(* IEC 61131-3 sources: MotionTestBenchMaster/Logical/02_HMI/HMI, 4 files *)

(* ---- Counter_Mng.st ---- *)
ACTION HMI_CounterInit:
	HMI_CounterCfgPartial.MachineCounters.HmiData[FillerLaps].Description				:= '@CounterDescription_001';
	HMI_CounterCfgPartial.MachineCounters.HmiData[ClosingUnit1Laps].Description			:= '@CounterDescription_002';
	HMI_CounterCfgPartial.MachineCounters.HmiData[ClosingUnit2Laps].Description			:= '@CounterDescription_003';
	HMI_CounterCfgPartial.MachineCounters.HmiData[RinserLaps].Description				:= '@CounterDescription_004';
	HMI_CounterCfgPartial.MachineCounters.HmiData[FlaworDoserLaps].Description			:= '@CounterDescription_005';
	HMI_CounterCfgPartial.MachineCounters.HmiData[PulpDoserLaps].Description			:= '@CounterDescription_006';
	HMI_CounterCfgPartial.MachineCounters.HmiData[PowerOn].Description					:= '@CounterDescription_007';

	HMI_CounterCfgPartial.ContainersCounters.HmiData[FillingFault].Description			:= '@CounterDescription_008';
	HMI_CounterCfgPartial.ContainersCounters.HmiData[FillingBurst].Description			:= '@CounterDescription_009';
	HMI_CounterCfgPartial.ContainersCounters.HmiData[ClosingUnit1Fault].Description		:= '@CounterDescription_010';
	HMI_CounterCfgPartial.ContainersCounters.HmiData[ClosingUnit2Fault].Description		:= '@CounterDescription_011';
	HMI_CounterCfgPartial.ContainersCounters.HmiData[RinsingFault].Description			:= '@CounterDescription_012';
	HMI_CounterCfgPartial.ContainersCounters.HmiData[PulpDoserFault].Description		:= '@CounterDescription_013';
	HMI_CounterCfgPartial.ContainersCounters.HmiData[FlaworDoserFault].Description		:= '@CounterDescription_014';
	HMI_CounterCfgPartial.ContainersCounters.HmiData[BurstEjected].Description			:= '@CounterDescription_015';
	HMI_CounterCfgPartial.ContainersCounters.HmiData[ManualEjected].Description			:= '@CounterDescription_016';
	HMI_CounterCfgPartial.ContainersCounters.HmiData[LowFillingEjected].Description		:= '@CounterDescription_017';
	HMI_CounterCfgPartial.ContainersCounters.HmiData[NotFilledEjected].Description		:= '@CounterDescription_018';
	HMI_CounterCfgPartial.ContainersCounters.HmiData[ContainersEntered].Description		:= '@CounterDescription_019';
	HMI_CounterCfgPartial.ContainersCounters.HmiData[ContainersProduced].Description	:= '@CounterDescription_020';
	HMI_CounterCfgPartial.ContainersCounters.HmiData[EjectionBySIS].Description			:= '@CounterDescription_045'; //V4.A.A.1.6.8
	HMI_CounterCfgPartial.ContainersCounters.HmiData[SIS_EjectionToBlower].Description			 := '@CounterDescription_046'; //V4.A.A.1.6.8
	HMI_CounterCfgPartial.ContainersCounters.HmiData[SIS_ContainersProducedToBlower].Description := '@CounterDescription_047'; //V4.A.A.1.6.8

	HMI_CounterCfgPartial.ProcessCounters.HmiData[FillerProduction].Description			:= '@CounterDescription_021';
	HMI_CounterCfgPartial.ProcessCounters.HmiData[ClosingUnit1Production].Description	:= '@CounterDescription_022';
	HMI_CounterCfgPartial.ProcessCounters.HmiData[ClosingUnit2Production].Description	:= '@CounterDescription_023';
	HMI_CounterCfgPartial.ProcessCounters.HmiData[RinserProduction].Description			:= '@CounterDescription_024';
	HMI_CounterCfgPartial.ProcessCounters.HmiData[PulpDoserProduction].Description		:= '@CounterDescription_025';
	HMI_CounterCfgPartial.ProcessCounters.HmiData[FlaworDoserProduction].Description	:= '@CounterDescription_026';
	HMI_CounterCfgPartial.ProcessCounters.HmiData[Cop].Description						:= '@CounterDescription_027';
	HMI_CounterCfgPartial.ProcessCounters.HmiData[FillerCip].Description				:= '@CounterDescription_044';
	HMI_CounterCfgPartial.ProcessCounters.HmiData[ClosingUnit1Cip].Description			:= '@CounterDescription_028';
	HMI_CounterCfgPartial.ProcessCounters.HmiData[ClosingUnit2Cip].Description			:= '@CounterDescription_029';
	HMI_CounterCfgPartial.ProcessCounters.HmiData[RinserCip].Description				:= '@CounterDescription_030';
	HMI_CounterCfgPartial.ProcessCounters.HmiData[PulpDoserCip].Description				:= '@CounterDescription_031';
	HMI_CounterCfgPartial.ProcessCounters.HmiData[FlaworDoserCip].Description			:= '@CounterDescription_032';

	HMI_CounterCfgPartial.EcoCounters.HmiData[Power].Description						:= '@CounterDescription_033';
	HMI_CounterCfgPartial.EcoCounters.HmiData[Air].Description							:= '@CounterDescription_034';
	HMI_CounterCfgPartial.EcoCounters.HmiData[GeneralCO2].Description					:= '@CounterDescription_035';
	HMI_CounterCfgPartial.EcoCounters.HmiData[ClosingUnitCO2].Description				:= '@CounterDescription_036';
	HMI_CounterCfgPartial.EcoCounters.HmiData[N2].Description							:= '@CounterDescription_037';
	HMI_CounterCfgPartial.EcoCounters.HmiData[ProcessWater].Description					:= '@CounterDescription_038';
	HMI_CounterCfgPartial.EcoCounters.HmiData[CopWater].Description						:= '@CounterDescription_039';
	HMI_CounterCfgPartial.EcoCounters.HmiData[BottomBottleCoolingWater].Description		:= '@CounterDescription_040';
	HMI_CounterCfgPartial.EcoCounters.HmiData[Product].Description						:= '@CounterDescription_041';
	HMI_CounterCfgPartial.EcoCounters.HmiData[Steam].Description						:= '@CounterDescription_042';
	HMI_CounterCfgPartial.EcoCounters.HmiData[FoodSteam].Description					:= '@CounterDescription_043';
	HMI_CounterCfgPartial.EcoCounters.HmiData[ProductWater].Description					:= '@CounterDescription_049'; //V4.A.A.1.6.14k
	HMI_CounterCfgPartial.EcoCounters.HmiData[Syrup].Description						:= '@CounterDescription_050'; //V4.A.A.1.6.14k

	HMI_CounterCfgPartial.EcoCounters.HmiData[Power].Unit								:= '';
	HMI_CounterCfgPartial.EcoCounters.HmiData[Air].Unit									:= '';
	HMI_CounterCfgPartial.EcoCounters.HmiData[GeneralCO2].Unit							:= '';
	HMI_CounterCfgPartial.EcoCounters.HmiData[ClosingUnitCO2].Unit						:= '';
	HMI_CounterCfgPartial.EcoCounters.HmiData[N2].Unit									:= '';
	HMI_CounterCfgPartial.EcoCounters.HmiData[ProcessWater].Unit						:= '';
	HMI_CounterCfgPartial.EcoCounters.HmiData[CopWater].Unit							:= '';
	HMI_CounterCfgPartial.EcoCounters.HmiData[BottomBottleCoolingWater].Unit			:= '';
	HMI_CounterCfgPartial.EcoCounters.HmiData[Product].Unit								:= '';
	HMI_CounterCfgPartial.EcoCounters.HmiData[Steam].Unit								:= '';
	HMI_CounterCfgPartial.EcoCounters.HmiData[FoodSteam].Unit							:= '';
	HMI_CounterCfgPartial.EcoCounters.HmiData[ProductWater].Unit						:= ''; //V4.A.A.1.6.14k
	HMI_CounterCfgPartial.EcoCounters.HmiData[Syrup].Unit								:= ''; //V4.A.A.1.6.14k
END_ACTION

ACTION HMI_CounterMng:
	CASE HMI_CounterPageCategory OF
		0:
			HMI_CounterPartialCfgPageDB		ACCESS	(ADR(HMI_CounterCfgPartial.MachineCounters));
			HMI_CounterPartialDataPageDB	ACCESS	(ADR(HMI_CounterDataPartial.MachineCounters));
			HMI_CounterTotalCfgPageDB		ACCESS	(ADR(HMI_CounterCfgTotal.MachineCounters));
			HMI_CounterTotalDataPageDB		ACCESS	(ADR(HMI_CounterDataTotal.MachineCounters));

		10:
			HMI_CounterPartialCfgPageDB		ACCESS	(ADR(HMI_CounterCfgPartial.ContainersCounters));
			HMI_CounterPartialDataPageDB	ACCESS	(ADR(HMI_CounterDataPartial.ContainersCounters));
			HMI_CounterTotalCfgPageDB		ACCESS	(ADR(HMI_CounterCfgTotal.ContainersCounters));
			HMI_CounterTotalDataPageDB		ACCESS	(ADR(HMI_CounterDataTotal.ContainersCounters));

		20:
			HMI_CounterPartialCfgPageDB		ACCESS	(ADR(HMI_CounterCfgPartial.ProcessCounters));
			HMI_CounterPartialDataPageDB	ACCESS	(ADR(HMI_CounterDataPartial.ProcessCounters));
			HMI_CounterTotalCfgPageDB		ACCESS	(ADR(HMI_CounterCfgTotal.ProcessCounters));
			HMI_CounterTotalDataPageDB		ACCESS	(ADR(HMI_CounterDataTotal.ProcessCounters));

		30:
			HMI_CounterPartialCfgPageDB		ACCESS	(ADR(HMI_CounterCfgPartial.EcoCounters));
			HMI_CounterPartialDataPageDB	ACCESS	(ADR(HMI_CounterDataPartial.EcoCounters));
			HMI_CounterTotalCfgPageDB		ACCESS	(ADR(HMI_CounterCfgTotal.EcoCounters));
			HMI_CounterTotalDataPageDB		ACCESS	(ADR(HMI_CounterDataTotal.EcoCounters));
	END_CASE

	HMI_TotalBottleProduced	:= HMI_CounterDataTotal.ContainersCounters.CounterData[ContainersProduced].CounterValue;

	//DATA TO EXCHANGE IN HMI WITH BLOWER //V4.A.A.1.7.0
	HMI_CounterHome.SS2P.Visibility 	:= CFG_Par.Machine.Combi.BLF OR CFG_Par.Machine.Combi.BAF;
	HMI_CounterHome.SS2P.Enable			:= CFG_Par.Machine.Combi.BLF OR CFG_Par.Machine.Combi.BAF;
	HMI_CounterHome.SS2P.LampON 		:= HMI_CounterHome.SS2P.ON;
	HMI_CounterHome.CounterValue[0] 	:= MAX(0,HMI_CounterDataPartial.ContainersCounters.CounterData[SIS_ContainersProducedToBlower].CounterValue -
													HMI_CounterDataPartial.ContainersCounters.CounterData[SIS_EjectionToBlower].CounterValue);
	HMI_CounterHome.CounterValue[1]		:= HMI_CounterDataPartial.ContainersCounters.CounterData[SIS_EjectionToBlower].CounterValue;

END_ACTION

(* ---- HMI_Init_CFG.st ---- *)
PROGRAM _INIT
	//AID
	HMI_AID_Loading;

	//ALR - Alarm
	HMI_ALR_Loading;

	//BTC - Bottles Bottom Cooling
	HMI_BTC_Loading;

	//CAP - Capper
	HMI_CAP_Loading;

	//CRW - Crowner
	HMI_CRW_Loading;

	// CO - Change Over
	HMI_CO_Loading;

	//COP - Cleaning out place
	HMI_COP_Loading;

	//CSR - Container Size Regulation
	HMI_CSR_Loading;

	//DMC - Dummy containers
	HMI_DMC_Loading;

	//GNS - General safety
	HMI_GNS_Loading;

	//MAU - Machine auxiliary
	HMI_MAU_Loading;

	//MNM - Main drive
	HMI_MNM_Loading;

	//MNT - Maintenance
	HMI_MNT_Loading;

	//ICO - Intelli Change Over
	HMI_ICO_Loading;

	//ITC - Interchange
	HMI_ITC_Loading;

	//OPS - Operator safety
	HMI_OPS_Loading;

	//HMI - Option Page
	HMI_OPT_Loading;

	//PAO - HMI PAO Page
	HMI_PAO_Loading;

	//RNS - RINSER
	HMI_RNS_Loading;

	//SFT - SHIFT REGISTER
	HMI_SFT_Loading;

	//TNK - Tank
	HMI_TNK_Loading;

	//Device (Valves - Instruments - Pumps)
	HMI_Valves_Loading;
	HMI_Instruments_Loading;
	HMI_Pumps_Loading;

	//HMI Variables
	HMI_Variables_Loading;

	HMI_CounterInit;
END_PROGRAM

(* ---- ITC_Mng.st ---- *)
ACTION HMI_ITCMng:
	IF HMI_ITC_Page.PartnerID <> HMI_ITC_PartnerOld OR NOT HMI_ITC_Partner_CFG[HMI_ITC_Page.PartnerID] THEN
		HMI_ITC_Page.PartnerID	:= LIMIT(CST_MinITCPartner, HMI_ITC_Page.PartnerID, CST_MaxITCPartner);
		FOR VAR_ITCindex := HMI_ITC_Page.PartnerID TO CST_MaxITCPartner DO
			IF HMI_ITC_Partner_CFG[VAR_ITCindex] THEN
				HMI_ITC_Page.PartnerID := VAR_ITCindex;
				EXIT;
			END_IF
		END_FOR

		HMI_ITC_Page.PageNum	:= 0;
		HMI_ITC_PartnerOld		:= HMI_ITC_Page.PartnerID;
		HMI_ITC_PageData.PageUp.Enable		:= FALSE;
		HMI_ITC_PageData.PageDown.Enable	:= FALSE;
	END_IF

	HMI_ITC_PageData ACCESS (ADR(HMI_ITC_PageDB[CST_MinITCPartner]) + MIN(HMI_ITC_Page.PartnerID - CST_MinITCPartner, CST_MaxITCPartner) * SIZEOF(HMI_ITC_PageDB[CST_MinITCPartner]));

	HMI_ITC_PageData.PageUp.LampON		:= HMI_ITC_PageData.PageUp.ON AND HMI_ITC_PageData.PageUp.Enable;
	HMI_ITC_PageData.PageDown.LampON	:= HMI_ITC_PageData.PageDown.ON AND HMI_ITC_PageData.PageDown.Enable;

	IF EDGEPOS(HMI_ITC_PageData.PageUp.LampON) THEN
		HMI_ITC_Page.PageNum	:= LIMIT(0, HMI_ITC_Page.PageNum + 1, 20);
		HMI_ITC_PageData.PageUp.Enable		:= FALSE;
		HMI_ITC_PageData.PageDown.Enable	:= FALSE;
	END_IF

	IF EDGEPOS(HMI_ITC_PageData.PageDown.LampON) THEN
		HMI_ITC_Page.PageNum	:= LIMIT(0, HMI_ITC_Page.PageNum - 1, 20);
		HMI_ITC_PageData.PageDown.Enable	:= FALSE;
		HMI_ITC_PageData.PageUp.Enable		:= FALSE;
	END_IF
END_ACTION

(* ---- Variables.var ---- *)
VAR
	HMI_ITC_PageData : REFERENCE TO HMI_ITC_Data_Type;
	HMI_ITC_PartnerOld : USINT;
	VAR_CoupledModality : SR := (Q1:=TRUE);
	VAR_BlrCombiModality : SR;
	VAR_LbrCombiModality : SR;
	VAR_ActCombiModality : SR; (*V4.A.A.1.6.12*)
	VAR_ContUnblock1 : SR;
	VAR_ContUnblock2 : SR;
	VAR_ContBlock1 : SR;
	VAR_ContBlock2 : SR;
	TMR_TON_WatchDogOn : TON;
	TMR_TON_WatchDogOff : TON;
	VAR_Temp_HmiPartnerID : USINT;
	VAR_ITCindex : USINT;
	RCPType_APCO : REAL;
	VAR_CoTypeOfChangeCFG : INT;
	HMI_CounterPartialDataPageDB : REFERENCE TO ARRAY[0..15] OF Counters_Type;
	HMI_CounterPartialCfgPageDB : REFERENCE TO ARRAY[0..15] OF HmiCounterData_Type;
	HMI_CounterTotalDataPageDB : REFERENCE TO ARRAY[0..15] OF Counters_Type;
	HMI_CounterTotalCfgPageDB : REFERENCE TO ARRAY[0..15] OF HmiCounterData_Type;
	HMI_CounterPageCategory : USINT;
	HMI_WatchDog : BOOL;
	VAR_BlrCombiModalityReset : BOOL; (*V4.A.A.1.6.12h*)
	VAR_SafetyVersionTemp : USINT; (*V4.A.A.1.6.13*)
	VAR_SafetyVersionData1 : STRING[2] := '0'; (*V4.A.A.1.6.13*)
	VAR_SafetyVersionData2 : STRING[2] := '0'; (*V4.A.A.1.6.13*)
	VAR_SafetyVersionData3 : STRING[2] := '0'; (*V4.A.A.1.6.13*)
	VAR_SafetyVersionData4 : STRING[2] := '0'; (*V4.A.A.1.6.13*)
END_VAR
